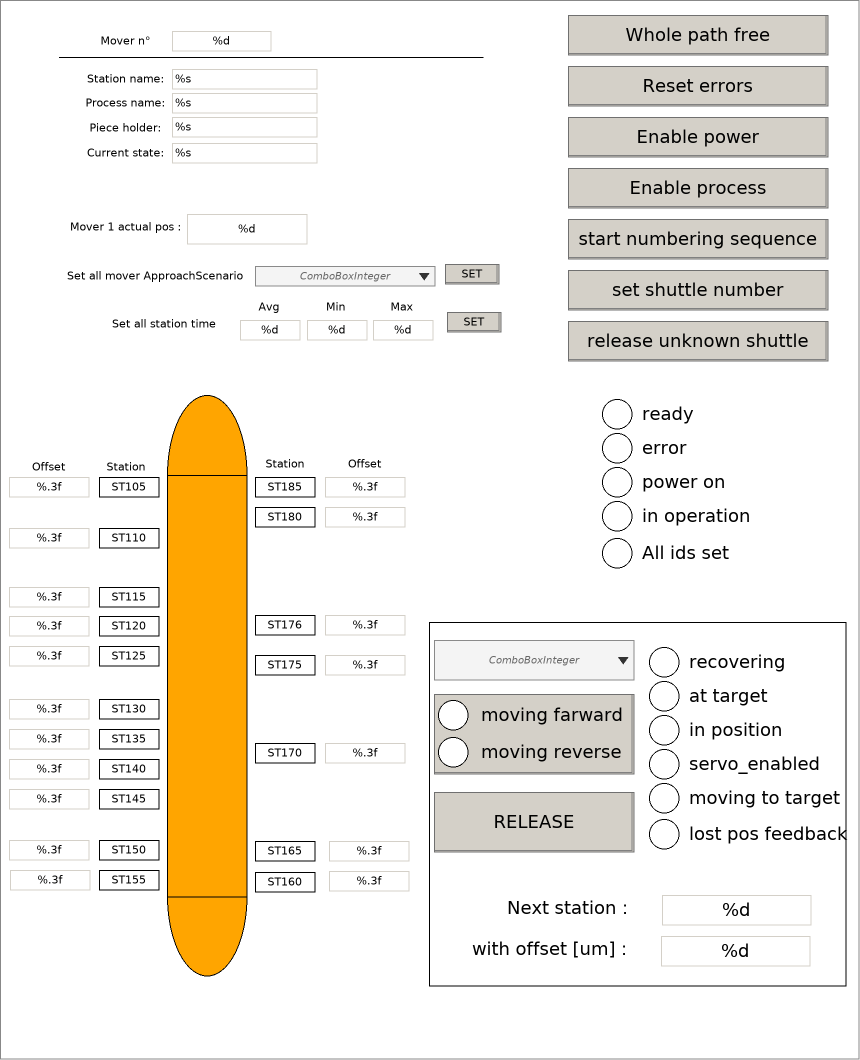
VISUALIZATION VISU_MoverDetail  // 860x1060
    Rectangle (429,622 417x364)
    Button (434,694 200x80)
        toggle gMoverAxis.Q_CT_Shuttle_to_BR.asStruct[HMI.selectedShuttle].bCommand.dirFarward
    Textfield (187,214 120x30), "%d", text variable: MAIN.MoverMan._MoverList[1]._MoverAxis._CurrentPos
        OnMouseDown: write the text variable via Default
    Label (38,212 146x30), "Mover 1 actual pos :"
    ComboBoxInteger (255,266 180x20), variable: MAIN.MoverMan.HMI_Scenario
    Label (59,261 187x30), "Set all mover ApproachScenario"
    Button (445,264 54x20), "SET"
        OnMouseDown: execute { MAIN.MoverMan.SetAllScenario(); }
    Label (93,309 126x30), "Set all station time"
    Textfield (240,320 60x20), "%d", text variable: MAIN.MoverMan.HMI_TimeAvg
        OnMouseDown: write the text variable via Default
    Label (241,296 56x22), "Avg"
    Textfield (307,320 60x20), "%d", text variable: MAIN.MoverMan.HMI_TimeMin
        OnMouseDown: write the text variable via Default
    Label (308,296 56x22), "Min"
    Textfield (373,320 60x20), "%d", text variable: MAIN.MoverMan.HMI_TimeMax
        OnMouseDown: write the text variable via Default
    Label (374,296 56x22), "Max"
    Button (447,312 54x20), "SET"
        OnMouseDown: execute { MAIN.MoverMan.SetAllTimers(ADR(PERS.iStationTimeDef1), 0); MAIN.MoverMan.SetAllTimers(ADR(PERS.iStationTimeDef2), 500); }
    Label (76,26 99x30), "Mover n°"
    Line (59,57) (483,57)
    Label (76,64 99x30), "Station name:"
    Label (76,88 99x30), "Process name:"
    Label (76,113 99x30), "Piece holder:"
    Label (76,138 99x30), "Current state:"
    Textfield (172,31 99x20), "%d", text variable: MAIN.MoverMan.HMI_iSelMover
        OnMouseDown: write the text variable via Default
    Textfield (172,69 145x20), "%s", text variable: MAIN.MoverMan._MoverList[MAIN.MoverMan.HMI_iSelMover].Station.ToString()
    Textfield (172,93 145x20), "%s"
    Textfield (172,117 145x20), "%s", text variable: MAIN.MoverMan._MoverList[MAIN.MoverMan.HMI_iSelMover].AttachedPieceHolder.ToString()
    Textfield (172,143 145x20), "%s", text variable: TO_STRING(MAIN.MoverMan._MoverList[MAIN.MoverMan.HMI_iSelMover]._State)
    Label (79,457 94x20), "Station"
    Label (-1,457 100x20), "Offset"
    Textfield (9,477 80x20), "%.3f", text variable: PERS.recipeList[PERS.iRecipeCurrent].stationOffsets[0]
        OnMouseDown: write the text variable via Default
    Textfield (9,528 80x20), "%.3f", text variable: PERS.recipeList[PERS.iRecipeCurrent].stationOffsets[1]
        OnMouseDown: write the text variable via Default
    Textfield (9,587 80x20), "%.3f", text variable: PERS.recipeList[PERS.iRecipeCurrent].stationOffsets[2]
        OnMouseDown: write the text variable via Default
    Textfield (9,616 80x20), "%.3f", text variable: PERS.recipeList[PERS.iRecipeCurrent].stationOffsets[3]
        OnMouseDown: write the text variable via Default
    Textfield (9,646 80x20), "%.3f", text variable: PERS.recipeList[PERS.iRecipeCurrent].stationOffsets[4]
        OnMouseDown: write the text variable via Default
    Textfield (9,699 80x20), "%.3f", text variable: PERS.recipeList[PERS.iRecipeCurrent].stationOffsets[5]
        OnMouseDown: write the text variable via Default
    Textfield (9,729 80x20), "%.3f", text variable: PERS.recipeList[PERS.iRecipeCurrent].stationOffsets[6]
        OnMouseDown: write the text variable via Default
    Textfield (9,759 80x20), "%.3f", text variable: PERS.recipeList[PERS.iRecipeCurrent].stationOffsets[7]
        OnMouseDown: write the text variable via Default
    Textfield (9,789 80x20), "%.3f", text variable: PERS.recipeList[PERS.iRecipeCurrent].stationOffsets[8]
        OnMouseDown: write the text variable via Default
    Textfield (9,840 80x20), "%.3f", text variable: PERS.recipeList[PERS.iRecipeCurrent].stationOffsets[9]
        OnMouseDown: write the text variable via Default
    Label (315,454 100x20), "Offset"
    Textfield (10,870 80x20), "%.3f", text variable: PERS.recipeList[PERS.iRecipeCurrent].stationOffsets[10]
        OnMouseDown: write the text variable via Default
    Textfield (325,477 80x20), "%.3f", text variable: PERS.recipeList[PERS.iRecipeCurrent].stationOffsets[17]
        OnMouseDown: write the text variable via Default
    Textfield (325,507 80x20), "%.3f", text variable: PERS.recipeList[PERS.iRecipeCurrent].stationOffsets[16]
        OnMouseDown: write the text variable via Default
    Textfield (325,615 80x20), "%.3f", text variable: PERS.recipeList[PERS.iRecipeCurrent].stationOffsets[15]
        OnMouseDown: write the text variable via Default
    Textfield (325,655 80x20), "%.3f", text variable: PERS.recipeList[PERS.iRecipeCurrent].stationOffsets[14]
        OnMouseDown: write the text variable via Default
    Textfield (325,743 80x20), "%.3f", text variable: PERS.recipeList[PERS.iRecipeCurrent].stationOffsets[13]
        OnMouseDown: write the text variable via Default
    Textfield (329,841 80x20), "%.3f", text variable: PERS.recipeList[PERS.iRecipeCurrent].stationOffsets[12]
        OnMouseDown: write the text variable via Default
    Textfield (329,871 80x20), "%.3f", text variable: PERS.recipeList[PERS.iRecipeCurrent].stationOffsets[11]
        OnMouseDown: write the text variable via Default
    Rectangle (99,870 60x20), "ST155", colour toggle: NOT GVL.st155_aut.xMoverPathFree
    Rectangle (99,840 60x20), "ST150", colour toggle: NOT GVL.st150_aut.xMoverPathFree
    Rectangle (99,789 60x20), "ST145", colour toggle: NOT GVL.st145_aut.xMoverPathFree
    Rectangle (99,759 60x20), "ST140", colour toggle: NOT GVL.st140_aut.xMoverPathFree
    Rectangle (99,729 60x20), "ST135", colour toggle: NOT GVL.st135_aut.xMoverPathFree
    Rectangle (99,699 60x20), "ST130", colour toggle: NOT GVL.st130_aut.xMoverPathFree
    Rectangle (99,646 60x20), "ST125", colour toggle: NOT GVL.st125_aut.xMoverPathFree
    Rectangle (99,616 60x20), "ST120", colour toggle: NOT GVL.st120_aut.xMoverPathFree
    Rectangle (99,587 60x20), "ST115", colour toggle: NOT GVL.st115_aut.xMoverPathFree
    Rectangle (99,528 60x20), "ST110", colour toggle: NOT GVL.st110_aut.xMoverPathFree
    Rectangle (99,477 60x20), "ST105", colour toggle: NOT GVL.st105_aut.xMoverPathFree
    Rectangle (255,507 60x20), "ST180", colour toggle: NOT GVL.st180_aut.xMoverPathFree
    Rectangle (255,615 60x20), "ST176", colour toggle: NOT GVL.st176_aut.xMoverPathFree
    Rectangle (255,655 60x20), "ST175", colour toggle: NOT GVL.st175_aut.xMoverPathFree
    Rectangle (255,743 60x20), "ST170", colour toggle: NOT GVL.st170_aut.xMoverPathFree
    Rectangle (255,841 60x20), "ST165", colour toggle: NOT GVL.st165_aut.xMoverPathFree
    Rectangle (255,872 60x20), "ST160", colour toggle: NOT GVL.st160_aut.xMoverPathFree
    Rectangle (255,477 60x20), "ST185", colour toggle: NOT GVL.st185_aut.xMoverPathFree
    Label (238,454 94x20), "Station"
    Ellipse (167,816 80x160)
    Ellipse (167,395 80x160)
    Rectangle (167,475 80x422)
    Button (568,66 260x40), "Reset errors"
        tap gMoverAxis.Q_CT_Track_to_BR.asStruct.bCommand.resetErrors
    Button (568,117 260x40), "Enable power"
        toggle gMoverAxis.Q_CT_Track_to_BR.asStruct.bCommand.enablePower
    ComboBoxInteger (434,640 200x40), variable: HMI.selectedShuttle
    Button (434,792 200x60), "RELEASE"
        tap gMoverAxis.Q_CT_Shuttle_to_BR.asStruct[HMI.selectedShuttle].bCommand.release
    Ellipse (649,647 30x30), colour toggle: gMoverAxis.I_CT_Shuttle_from_BR.asStruct[HMI.selectedShuttle].bStatus.recovering
    Label (686,647 160x30), "recovering"
    Ellipse (649,681 30x30), colour toggle: gMoverAxis.I_CT_Shuttle_from_BR.asStruct[HMI.selectedShuttle].bStatus.at_target
    Label (686,681 160x30), "at target"
    Ellipse (649,715 30x30), colour toggle: gMoverAxis.I_CT_Shuttle_from_BR.asStruct[HMI.selectedShuttle].bStatus.in_position
    Label (686,715 160x30), "in position"
    Ellipse (649,749 30x30), colour toggle: gMoverAxis.I_CT_Shuttle_from_BR.asStruct[HMI.selectedShuttle].bStatus.servo_enabled
    Label (686,749 160x30), "servo_enabled"
    Ellipse (649,783 30x30), colour toggle: gMoverAxis.I_CT_Shuttle_from_BR.asStruct[HMI.selectedShuttle].bStatus.moving_to_load_target
    Label (686,783 160x30), "moving to target"
    Ellipse (649,819 30x30), colour toggle: gMoverAxis.I_CT_Shuttle_from_BR.asStruct[HMI.selectedShuttle].bStatus.lost_position_feedback
    Label (686,819 160x30), "lost pos feedback"
    Ellipse (602,399 30x30), colour toggle: gMoverAxis.I_CT_Track_from_BR.asStruct.bStatus.ready
    Label (639,399 160x30), "ready"
    Ellipse (602,433 30x30), colour toggle: gMoverAxis.I_CT_Track_from_BR.asStruct.bStatus.error
    Label (639,433 160x30), "error"
    Ellipse (602,467 30x30), colour toggle: gMoverAxis.I_CT_Track_from_BR.asStruct.bStatus.powerOn
    Label (639,467 160x30), "power on"
    Ellipse (602,501 30x30), colour toggle: gMoverAxis.I_CT_Track_from_BR.asStruct.bStatus.inOperation
    Label (639,501 160x30), "in operation"
    Button (568,168 260x40), "Enable process"
        toggle gMoverAxis.Q_CT_Track_to_BR.asStruct.bCommand.enableProcess
    Button (568,219 260x40), "start numbering sequence"
        toggle gMoverAxis.Q_CT_Track_to_BR.asStruct.bCommand.startMoverNumberingSequence
    Button (568,270 260x40), "set shuttle number"
        tap gMoverAxis.Q_CT_Track_to_BR.asStruct.bCommand.setShuttleNumber
    Button (568,321 260x40), "release unknown shuttle"
        tap gMoverAxis.Q_CT_Track_to_BR.asStruct.bCommand.releaseUnknownShuttle
    Ellipse (438,700 30x30), colour toggle: gMoverAxis.Q_CT_Shuttle_to_BR.asStruct[HMI.selectedShuttle].bCommand.dirFarward
    Ellipse (438,737 30x30), colour toggle: NOT gMoverAxis.Q_CT_Shuttle_to_BR.asStruct[HMI.selectedShuttle].bCommand.dirFarward
    Label (478,700 160x30), "moving farward"
    Label (478,737 160x30), "moving reverse"
    Button (568,15 260x40), "Whole path free"
        toggle gMoverAxis.Q_CT_Track_to_BR.asStruct.bCommand.wholePathFree
    Textfield (662,895 149x30), "%d", text variable: gMoverAxis.Q_CT_Shuttle_to_BR.asStruct[HMI.selectedShuttle].bNextStation
        OnMouseDown: write the text variable via Default
    Label (471,893 160x30), "Next station :"
    Textfield (661,936 149x30), "%d", text variable: gMoverAxis.Q_CT_Shuttle_to_BR.asStruct[HMI.selectedShuttle].diNextOffset_um
        OnMouseDown: write the text variable via Default
    Label (470,934 160x30), "with offset [um] :"
    Ellipse (602,538 30x30), colour toggle: gMoverAxis.I_CT_Track_from_BR.asStruct.bStatus.allIdSet
    Label (639,538 160x30), "All ids set"
END_VISUALIZATION

(* stored: Version 1.1.0.1, ProductVersion 3.1.4024.6
   Visu VISU_MoverDetail: Id {3c60e503-48c2-4a6b-81a1-aaecffae9186} *)
